# EPICS autosave request: iocBoot/iocdmm7510/auto_settings_dcct.req
file "dcct_settings.req",                P=$(P),  R=$(R)
file "dmm7510_settings.req",             P=$(P),  R=$(R)
